FUNCTION_BLOCK CRANE_1_SUBSCRIBE (* Composite Function Block Type *)
  (* Standard: 61499-2 *)
  (* Version 1.0, 2019-04-13, adeel *)
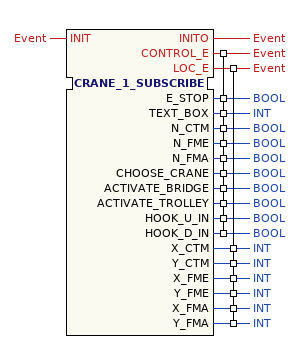
  EVENT_INPUT
    INIT; (* Initialization Request *)
  END_EVENT
  EVENT_OUTPUT
    INITO; (* Initialization Confirm *)
    CONTROL_E WITH E_STOP, TEXT_BOX, N_CTM, N_FME, N_FMA, CHOOSE_CRANE, ACTIVATE_BRIDGE, ACTIVATE_TROLLEY, HOOK_U_IN, HOOK_D_IN; (* Execution Confirmation *)
    LOC_E WITH X_CTM, Y_CTM, X_FME, Y_FME, X_FMA, Y_FMA;
  END_EVENT
  VAR_OUTPUT
    E_STOP : BOOL;
    TEXT_BOX : INT;
    N_CTM : BOOL;
    N_FME : BOOL;
    N_FMA : BOOL;
    CHOOSE_CRANE : BOOL;
    ACTIVATE_BRIDGE : BOOL;
    ACTIVATE_TROLLEY : BOOL;
    HOOK_U_IN : BOOL;
    HOOK_D_IN : BOOL;
    X_CTM : INT;
    Y_CTM : INT;
    X_FME : INT;
    Y_FME : INT;
    X_FMA : INT;
    Y_FMA : INT;
  END_VAR
  FBS
    SUBSCRIBE_1 : SUBSCRIBE_1(QI := 1, ID := opc_ua[/Objects/1:CRANE1A]);
    SUBSCRIBE_1_1 : SUBSCRIBE_1(QI := 1, ID := opc_ua[/Objects/1:CRANE1B]);
    SUBSCRIBE_1_2 : SUBSCRIBE_1(QI := 1, ID := opc_ua[/Objects/1:CRANE1C]);
    SUBSCRIBE_1_3 : SUBSCRIBE_1(QI := 1, ID := opc_ua[/Objects/1:CRANE1D]);
    SUBSCRIBE_1_4 : SUBSCRIBE_1(QI := 1, ID := opc_ua[/Objects/1:CRANE1E]);
    SUBSCRIBE_1_5 : SUBSCRIBE_1(QI := 1, ID := opc_ua[/Objects/1:CRANE1F]);
    SUBSCRIBE_1_6 : SUBSCRIBE_1(QI := 1, ID := opc_ua[/Objects/1:CRANE1G]);
    SUBSCRIBE_1_7 : SUBSCRIBE_1(QI := 1, ID := opc_ua[/Objects/1:CRANE1H]);
    SUBSCRIBE_1_8 : SUBSCRIBE_1(QI := 1, ID := opc_ua[/Objects/1:CRANE1I]);
    SUBSCRIBE_1_9 : SUBSCRIBE_1(QI := 1, ID := opc_ua[/Objects/1:CRANE1J]);
    SUBSCRIBE_1_10 : SUBSCRIBE_1(QI := 1, ID := opc_ua[/Objects/1:CRANE1K]);
    SUBSCRIBE_1_11 : SUBSCRIBE_1(QI := 1, ID := opc_ua[/Objects/1:CRANE1L]);
    SUBSCRIBE_1_12 : SUBSCRIBE_1(QI := 1, ID := opc_ua[/Objects/1:CRANE1M]);
    SUBSCRIBE_1_13 : SUBSCRIBE_1(QI := 1, ID := opc_ua[/Objects/1:CRANE1N]);
    SUBSCRIBE_1_14 : SUBSCRIBE_1(QI := 1, ID := opc_ua[/Objects/1:CRANE1O]);
    SUBSCRIBE_1_15 : SUBSCRIBE_1(QI := 1, ID := opc_ua[/Objects/1:CRANE1P]);
    N_FMA : BOOL2BOOL;
    E_STOP : BOOL2BOOL;
    N_CTM : BOOL2BOOL;
    N_FME : BOOL2BOOL;
    TEXT_BOX : INT2INT;
    CHOOSE_CRANE : BOOL2BOOL;
    ACTIVATE_BRIDGE : BOOL2BOOL;
    X_CTM : INT2INT;
    ACTIVATE_TROLLEY : BOOL2BOOL;
    HOOK_U_IN : BOOL2BOOL;
    HOOK_D_IN : BOOL2BOOL;
    Y_CTM : INT2INT;
    X_FME : INT2INT;
    Y_FME : INT2INT;
    X_FMA : INT2INT;
    Y_FMA : INT2INT;
  END_FBS
  EVENT_CONNECTIONS
    SUBSCRIBE_1.INITO TO SUBSCRIBE_1_1.INIT;
    SUBSCRIBE_1_1.INITO TO SUBSCRIBE_1_2.INIT;
    SUBSCRIBE_1_2.INITO TO SUBSCRIBE_1_3.INIT;
    SUBSCRIBE_1_4.INITO TO SUBSCRIBE_1_5.INIT;
    SUBSCRIBE_1_5.INITO TO SUBSCRIBE_1_6.INIT;
    SUBSCRIBE_1_6.INITO TO SUBSCRIBE_1_7.INIT;
    SUBSCRIBE_1_7.INITO TO SUBSCRIBE_1_8.INIT;
    SUBSCRIBE_1_8.INITO TO SUBSCRIBE_1_9.INIT;
    SUBSCRIBE_1_9.INITO TO SUBSCRIBE_1_10.INIT;
    SUBSCRIBE_1_10.INITO TO SUBSCRIBE_1_11.INIT;
    SUBSCRIBE_1_11.INITO TO SUBSCRIBE_1_12.INIT;
    SUBSCRIBE_1_12.INITO TO SUBSCRIBE_1_13.INIT;
    SUBSCRIBE_1_13.INITO TO SUBSCRIBE_1_14.INIT;
    SUBSCRIBE_1_14.INITO TO SUBSCRIBE_1_15.INIT;
    INIT TO SUBSCRIBE_1.INIT;
    SUBSCRIBE_1_3.INITO TO SUBSCRIBE_1_4.INIT;
    SUBSCRIBE_1.IND TO E_STOP.REQ;
    SUBSCRIBE_1_1.IND TO TEXT_BOX.REQ;
    SUBSCRIBE_1_2.IND TO N_CTM.REQ;
    SUBSCRIBE_1_3.IND TO N_FME.REQ;
    E_STOP.CNF TO CONTROL_E;
    TEXT_BOX.CNF TO CONTROL_E;
    N_CTM.CNF TO CONTROL_E;
    N_FME.CNF TO CONTROL_E;
    SUBSCRIBE_1_4.IND TO N_FMA.REQ;
    N_FMA.CNF TO CONTROL_E;
    SUBSCRIBE_1_5.IND TO CHOOSE_CRANE.REQ;
    SUBSCRIBE_1_6.IND TO ACTIVATE_BRIDGE.REQ;
    SUBSCRIBE_1_7.IND TO ACTIVATE_TROLLEY.REQ;
    SUBSCRIBE_1_8.IND TO HOOK_U_IN.REQ;
    SUBSCRIBE_1_9.IND TO HOOK_D_IN.REQ;
    SUBSCRIBE_1_10.IND TO X_CTM.REQ;
    SUBSCRIBE_1_11.IND TO Y_CTM.REQ;
    SUBSCRIBE_1_12.IND TO X_FME.REQ;
    SUBSCRIBE_1_13.IND TO Y_FME.REQ;
    SUBSCRIBE_1_14.IND TO X_FMA.REQ;
    SUBSCRIBE_1_15.IND TO Y_FMA.REQ;
    CHOOSE_CRANE.CNF TO CONTROL_E;
    ACTIVATE_BRIDGE.CNF TO CONTROL_E;
    ACTIVATE_TROLLEY.CNF TO CONTROL_E;
    HOOK_U_IN.CNF TO CONTROL_E;
    HOOK_D_IN.CNF TO CONTROL_E;
    X_CTM.CNF TO LOC_E;
    Y_CTM.CNF TO LOC_E;
    X_FME.CNF TO LOC_E;
    Y_FME.CNF TO LOC_E;
    X_FMA.CNF TO LOC_E;
    Y_FMA.CNF TO LOC_E;
    SUBSCRIBE_1_15.INITO TO INITO;
  END_CONNECTIONS
  DATA_CONNECTIONS
    SUBSCRIBE_1.RD_1 TO E_STOP.IN;
    SUBSCRIBE_1_1.RD_1 TO TEXT_BOX.IN;
    SUBSCRIBE_1_2.RD_1 TO N_CTM.IN;
    SUBSCRIBE_1_3.RD_1 TO N_FME.IN;
    E_STOP.OUT TO E_STOP;
    TEXT_BOX.OUT TO TEXT_BOX;
    N_CTM.OUT TO N_CTM;
    N_FME.OUT TO N_FME;
    SUBSCRIBE_1_4.RD_1 TO N_FMA.IN;
    N_FMA.OUT TO N_FMA;
    SUBSCRIBE_1_5.RD_1 TO CHOOSE_CRANE.IN;
    SUBSCRIBE_1_6.RD_1 TO ACTIVATE_BRIDGE.IN;
    SUBSCRIBE_1_7.RD_1 TO ACTIVATE_TROLLEY.IN;
    SUBSCRIBE_1_8.RD_1 TO HOOK_U_IN.IN;
    SUBSCRIBE_1_9.RD_1 TO HOOK_D_IN.IN;
    SUBSCRIBE_1_10.RD_1 TO X_CTM.IN;
    SUBSCRIBE_1_11.RD_1 TO Y_CTM.IN;
    SUBSCRIBE_1_12.RD_1 TO X_FME.IN;
    SUBSCRIBE_1_13.RD_1 TO Y_FME.IN;
    SUBSCRIBE_1_14.RD_1 TO X_FMA.IN;
    SUBSCRIBE_1_15.RD_1 TO Y_FMA.IN;
    CHOOSE_CRANE.OUT TO CHOOSE_CRANE;
    HOOK_U_IN.OUT TO HOOK_U_IN;
    ACTIVATE_BRIDGE.OUT TO ACTIVATE_BRIDGE;
    ACTIVATE_TROLLEY.OUT TO ACTIVATE_TROLLEY;
    HOOK_D_IN.OUT TO HOOK_D_IN;
    X_CTM.OUT TO X_CTM;
    Y_CTM.OUT TO Y_CTM;
    X_FME.OUT TO X_FME;
    Y_FME.OUT TO Y_FME;
    X_FMA.OUT TO X_FMA;
    Y_FMA.OUT TO Y_FMA;
  END_CONNECTIONS
END_FUNCTION_BLOCK
